// TIA Portal V17 export
// export: Created 2025-06-26T07:49:16.1238182Z, ExportSetting WithDefaults, DisplayName Totally Integrated Automation Portal, DisplayVersion V17 Update 8, DisplayName TIA Portal Openness, DisplayVersion V17 Update 8, DisplayName TIA Portal Version Control Interface, DisplayVersion V17, DisplayName STEP 7 Professional, DisplayVersion V17 Update 8, DisplayName STEP 7 Safety, DisplayVersion V17 Update 6, DisplayName WinCC Advanced, DisplayVersion V17 Update 8
DATA_BLOCK "ModbusRTUMaster_DB"   // DB27
VERSION : 0.1
// stored: AutoNumber true, DBAccessibleFromOPCUA true, InstanceOfName ModbusRTUMaster, InstanceOfType FB
"ModbusRTUMaster"
   // VAR_INPUT
   //    bFirstCycle : Bool;
   //    bStart : Bool;
   // END_VAR
   // VAR_OUTPUT
   //    Done { ExternalAccessible := 'False'; ExternalVisible := 'False'; ExternalWritable := 'False'} : Bool;
   //    Initialised : Bool;
   // END_VAR
   // VAR
   //    InitReq : Bool;
   //    InitErrorCode : Word;
   //    InitSuccess : Bool;
   //    ReadReq : Bool;
   //    MasterDoneStored : Bool;
   //    MasterStatus_stored : Word;
   //    MasterDone : Bool;
   //    MasterError : Bool;
   //    MasterBusy : Bool;
   //    MasterStatus : Word;
   //    State : USInt;
   //    Wait : TON_TIME;
   //    Node1CommCycles { S7_SetPoint := 'True'} : UDInt;
   //    Node2CommCycles : UDInt;
   //    Node10CommCycles : UDInt;
   //    Node20CommCycles : UDInt;
   // END_VAR
BEGIN
END_DATA_BLOCK
